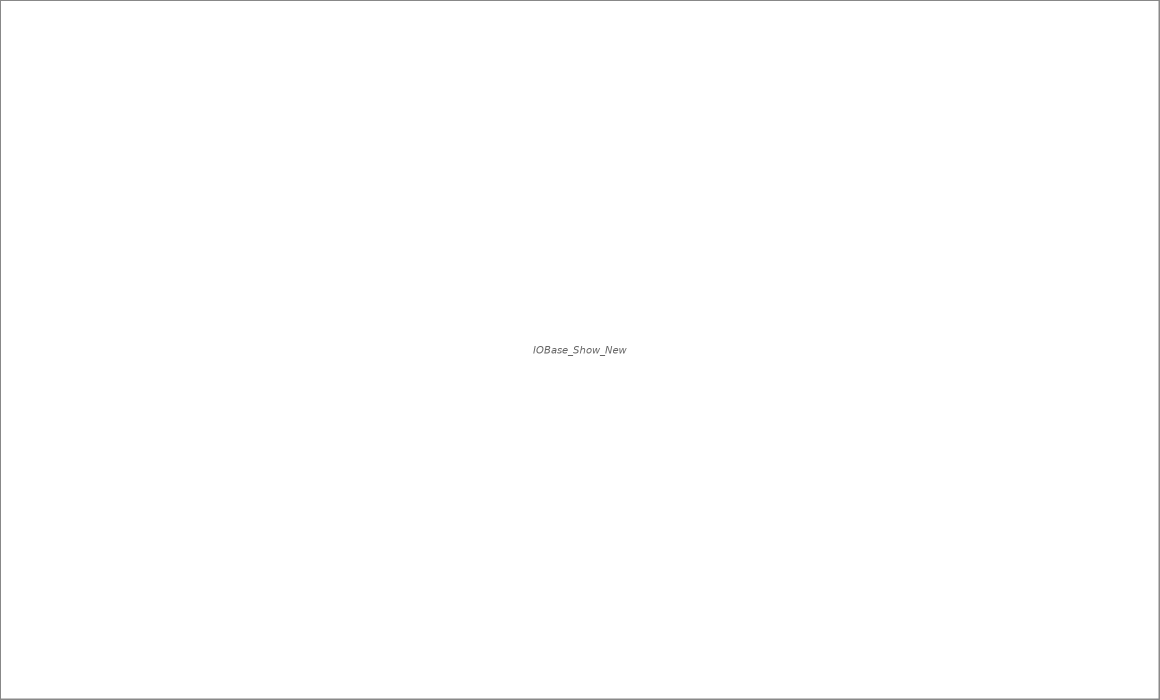
VISUALIZATION IO_Output  // 1160x700
    TabControl (0,0 1160x700)
        shows IOBase_Show_New(userData := TesterIO.fbIOBase_Output.HMIITF)
        [0]: TabTitle=Output
END_VISUALIZATION

(* stored: Version 1.1.0.1, ProductVersion 3.1.4024.4
   Visu IO_Output: Id {47e31e44-61ea-4d02-bc01-2d4d10a87944} *)
